(*	This FB is used for a single output solenoid 
	It uses the times to say when Extended/Retracted  	
	It starts assuming retracted and the output off.
*)
FUNCTION_BLOCK FB_GantryXYCylinder EXTENDS FB_ComponentBase IMPLEMENTS I_Cylinder
VAR
    //Output
    Output AT %Q* : BOOL;

    // Internal variables
    _ExtendRequest  : BOOL;
    _RetractRequest : BOOL;
    _Extended       : BOOL;
    _Retracted      : BOOL;
    _Extending      : BOOL;
    _Retracting     : BOOL;
    _ExtendTime     : LREAL := 1000; // Default time 1s
    _RetractTime    : LREAL := 1000; // Default time 1s

    // Timer for Extend/Retract
    Extend_TON    : TON;
    Retract_TON   : TON;
    Extend_RTRIG  : R_TRIG;
    Retract_RTRIG : R_TRIG;

    //HMI 
    Cylinder_HMI : ST_Cylinder_HMI;
END_VAR

METHOD PROTECTED CreateEvents
VAR_INPUT
END_VAR
SUPER^.CreateEvents();
END_METHOD

METHOD CyclicLogic
//One shot the requests
Extend_RTRIG(CLK := _ExtendRequest);
Retract_RTRIG(CLK := _RetractRequest);

//Handle Extend
IF Extend_RTRIG.Q THEN
    Output          := TRUE;
    _Extending      := TRUE;
    _Retracting     := FALSE;
    _Retracted      := FALSE;
    _RetractRequest := FALSE;
END_IF

//Handle Retract
IF Retract_RTRIG.Q THEN
    Output         := FALSE;
    _Extending     := FALSE;
    _Retracting    := TRUE;
    _Extended      := FALSE;
    _ExtendRequest := FALSE;
END_IF

//Handle the time to Extend/Retract
Extend_TON(IN := _Extending, PT := LREAL_TO_TIME(_ExtendTime));
Retract_TON(IN := _Retracting, PT := LREAL_TO_TIME(_RetractTime));
IF Extend_TON.Q THEN
    _Extended  := TRUE;
    _Extending := FALSE;
END_IF

IF Retract_TON.Q THEN
    _Retracted  := TRUE;
    _Retracting := FALSE;
END_IF

SUPER^.CyclicLogic();
END_METHOD

METHOD Extend
_ExtendRequest  := TRUE;
_RetractRequest := FALSE;
END_METHOD

PROPERTY Extended : BOOL
GET
Extended := _Extended;
END_GET
END_PROPERTY

PROPERTY ExtendTime : LREAL
GET
ExtendTime := _ExtendTime;
END_GET
SET
END_SET
END_PROPERTY

METHOD PROTECTED HMICommunication
VAR_INPUT
END_VAR
SUPER^.HMICommunication();

//Handle the requests to extend and retract
IF ComponentBase_HMI.Status.HMIControlAvailable THEN
    IF Cylinder_HMI.Command.Extend THEN
        Extend();
    ELSIF Cylinder_HMI.Command.Retract THEN
        Retract();
    END_IF
END_IF

//Update HMI status info
Cylinder_HMI.Status.Extended    := _Extended;
Cylinder_HMI.Status.Extending   := _Extending;
Cylinder_HMI.Status.Retracted   := _Retracted;
Cylinder_HMI.Status.Retracting  := _Retracting;
Cylinder_HMI.Config.ExtendTime  := _ExtendTime;
Cylinder_HMI.Config.RetractTime := _RetractTime;
END_METHOD

//! @summary Basic component initialization logic
METHOD PROTECTED Initialize : BOOL;

//! @description This method is called by <c>CyclicLogic()</c> as required
//Set the cylinder to retracted
IF Output THEN
    _Extended  := TRUE;
    _Retracted := FALSE;
ELSE
    _Extended  := FALSE;
    _Retracted := TRUE;
END_IF

_Extending      := FALSE;
_ExtendRequest  := FALSE;
_Retracting     := FALSE;
_RetractRequest := FALSE;

//Call base class Initialize
Initialize := SUPER^.Initialize();
END_METHOD

METHOD PROTECTED Monitoring
VAR_INPUT
END_VAR
_Busy    := _Extending OR _Retracting;
_Error   := FALSE;
_ErrorID := 0;
SUPER^.Monitoring();
END_METHOD

METHOD Retract
_ExtendRequest  := FALSE;
_RetractRequest := TRUE;
END_METHOD

PROPERTY Retracted : BOOL
GET
Retracted := _Retracted;
END_GET
END_PROPERTY

PROPERTY RetractTime : LREAL
GET
RetractTime := _RetractTime;
END_GET
SET
_RetractTime := RetractTime;
END_SET
END_PROPERTY

END_FUNCTION_BLOCK

(* stored: Version 1.1.0.1
   POU FB_GantryXYCylinder: Id {84ff1c9d-387b-40dd-9e52-4cc6c2a7141b}, SpecialFunc None
   Method CreateEvents: Id {3e5b5b40-936d-40ba-aba9-afaf2438d26e}
   Method CyclicLogic: Id {5c1b5fa3-af8d-4464-9679-0f6e0bdf420f}
   Method Extend: Id {f76b6140-af7b-4e84-89e2-4088b7535499}
   Property Extended: Id {0b637275-f326-40fc-9e85-9bc95eea83ca}
   Get Get: Id {0461fe63-f86f-44be-aaa4-3be89e903078}
   Property ExtendTime: Id {e2dcc71a-7531-40a4-928f-f19b69a1fb32}
   Get Get: Id {0b001083-9d94-4ade-8f8e-cfb190c4a6ef}
   Set Set: Id {776c832f-beb9-4f81-a446-99e1808f8b74}
   Method HMICommunication: Id {ecf4504c-d862-48e6-991f-2e1997844380}
   Method Initialize: Id {87e9fdf5-09e8-42e1-9c25-a88a111319f8}
   Method Monitoring: Id {9843f90f-d434-4d6f-8841-844359423366}
   Method Retract: Id {62f4be5a-2417-454d-83fa-0301d008b1f8}
   Property Retracted: Id {6d4508b6-aaa4-44e0-b03b-568180b910d9}
   Get Get: Id {c858b548-e496-44d8-871e-eecca4d05383}
   Property RetractTime: Id {e14f84fd-065d-441b-b8bd-492d5e46847d}
   Get Get: Id {04369b4b-f6ef-486b-bf2c-c677ad5bd77a}
   Set Set: Id {8b666dbf-e9ab-4b6d-a120-fcb12ea4f469} *)
